# EPICS StreamDevice protocol: agilent3631ASup/devagilent3631A.proto
getIDN {
    out "*IDN?";
    #Read no more that 39 chars (EPICS limit)
    in "%/(.{0,39})/";
    ExtraInput = Ignore;
}

read_current {
    out "MEAS:CURR?";
    in "%f";
	ExtraInput = Ignore;
}

write_current {
    out "CURR %f";
}

read_voltage {
    out "MEAS:VOLT?";
    in "%f";
	ExtraInput = Ignore;
}

write_voltage {
    out "VOLT %f";
}

read_output_status{
    out "OUTP?";
    in "%d";
	ExtraInput = Ignore;
}

write_output_status{
    out "OUTP %d";
}

read_error_status{
    out "SYST:ERR?";
    in "%s";
	ExtraInput = Ignore;
}

set_Local_Remote {
    out "SYST:%{LOC|REM}";
}
